# EPICS substitutions: CaenDigApp/Db/userHost.substitutions
# Example substitutions file

file "db/dbExample1.db" {
    { user = "epicsHost" }
}

file db/dbExample2.db {
    pattern { user, no, scan }
        { "epicsHost", 1, "1 second" }
        { "epicsHost", 2, "2 second" }
        { "epicsHost", 3, "5 second" }
}
